INTERFACE I_GroupBuilder

END_INTERFACE

(* stored: Version 1.1.0.1, ProductVersion 3.1.4024.12
   Itf I_GroupBuilder: Id {67e4f0d6-3ff4-4b2b-8fd7-8b7bc2c1c622} *)
